TYPE ST_BaseHMIControlElement_View :
STRUCT
	bDanaBaseControlElement		: BOOL;
	
END_STRUCT
END_TYPE

(* stored: Version 1.1.0.1
   DUT ST_BaseHMIControlElement_View: Id {eb9c7dc9-a2ac-0d87-200e-8ddc8d79ced0} *)
